(* Logix 5000 project; controller BTS01 vendor 1 type 14 code 217 rev 32.14; software revision 32.04; part 12 of 15 *)
(* tags used below, declared in another part *)
   ApplyDST : SINT;
   C02S03 : INT;   // 5069-IB16
   CAUSTIC_DRAIN_LATCH : BOOL;
   CAUSTIC_DRAIN_RUN : BOOL;
   CAUSTIC_DRAIN_RUN_CLR : BOOL;
   CAUSTIC_DRAIN_RUN_PB : BOOL;
   CAUSTIC_FILL_PB_HMI : BOOL;
   CAUSTIC_FILL_RUN : BOOL;
   CAUSTIC_FILL_RUN_CLR : BOOL;
   CAUSTIC_PREP_LATCH : BOOL;
   CAUSTIC_PREP_RUN : BOOL;
   CAUSTIC_PREP_RUN_CLR : BOOL;   // CAUSTIC PREP JKFF CLEAR BIT
   CAUSTIC_PREP_RUN_PB : BOOL;
   CAUSTIC_PREP_TEMP_SPT : REAL;
   CAUSTIC_PREP_TIME_SPT : REAL;
   CAUSTIC_TANK_LEVEL_OFF_PERC : DINT;   // HMI INPUT OF WATER LEVEL OFF IN %
   CIP1_CAUSTIC_DRAIN_FILE : DINT;   // CIP 1 RAW RECIEVING CIP CAUSTIC DRAIN ENABLE REFERENCE FILE
   CIP1_CAUSTIC_PREP_FILE : DINT;   // CIP 1 RAW RECIEVING CIP CAUSTIC PREP ENABLE REFERENCE FILE
   CIP1_FINALRINSE_DRAIN_FILE : DINT;   // CIP 1 RAW RECIEVING CIP FINAL RINSE DRAIN ENABLE REFERENCE FILE
   CIP1_PRERINSE_DRAIN_FILE : DINT;   // CIP 1 RAW RECIEVING CIP PRERINSE DRAIN ENABLE REFERENCE FILE
   CIP1_PRERINSE_PREP_FILE : DINT;   // CIP 1 RAW RECIEVING CIP PRERINSE PREP ENABLE REFERENCE FILE
   CIP_1_ACTIVE_STEP : CIP_STEP_DEF;   // CIP 1 ACTIVE STEP DATA
   CIP_1_ALARMS : DINT[30];
   CIP_1_AVAIL_STEP_ID : DINT;
   CIP_1_CAUSTIC_TRANS_ACT : BOOL;   // CIP 1 RETURN TO CAUSTIC TANK LEVEL TRANSITION ACTIVE
   CIP_1_CIRCUIT_SELECT_EDIT_HMI : INT;
   CIP_1_EDIT_PROGRAM : CIP_PROGRAM;
   CIP_1_INSERT_STEP : DINT;   // CIP1 INSERT STEP POINTER
   CIP_1_LOAD_RECIPE_EDIT_PB : BOOL;
   CIP_1_MASTER_REF_FILE : DINT[15,30];   // SEQUENCER PINS CIP 1
   CIP_1_PRERINSE_TRANS_ACT : BOOL;   // CIP 1 RETURN TO PRERINSE TANK LEVEL TRANSITION ACTIVE
   CIP_1_PRERINSE_TRANS_DRAIN : BOOL;   // CIP 1 RETURN TO PRERINSE TANK LEVEL TRANSITION ACTIVE
   CIP_1_PROGRAM_ID : INT;
   CIP_1_PROGRAMS : CIP_PROGRAM[30];
   CIP_1_RESET_PB_HMI : BOOL;
   CIP_1_RETURN_HMI : DINT;   // CIP 1 RETURN LOCATION HMI INDICATOR
   CIP_1_RETURN_TO_CAUSTIC : BOOL;   // CIP 1 RETURN TO CAUSTIC TANK DURING CAUSTIC RETURN STEPS
   CIP_1_RETURN_TO_PRERINSE : BOOL;   // CIP 1 RETURN TO PRE-RINSE TANK DURING CAUSTIC RETURN STEPS
   CIP_1_REVERT_RECIPE_EDITS_PB : BOOL;
   CIP_1_RUN_LATCH : BOOL;
   CIP_1_SAVE_RECIPE_EDITS_PB : BOOL;
   CIP_1_SEQ_CTU : COUNTER;   // CIP 1 SEQUENCE STEP COUNTER THIS IS THE SEQUENCE STEP CONTROL
   CIP_1_SEQ_ENABLE : DINT;   // CIP 1 SEQUENCER DATA TO BE ENABLED FOR OPERATION DURING CIP
   CIP_1_STEP_AVAIL_NAMES : CIP_STEP_DEF[30];
   CIP_1_STEP_COPY : BOOL;
   CIP_1_STEP_DELETE : BOOL;
   CIP_1_STEP_DELETING : BOOL;
   CIP_1_STEP_ID : INT;
   CIP_1_STEP_INSERT_PB : BOOL;   // CIP1 STEP INSERT PB FROM HMI
   CIP_1_STEP_INSERTING : BOOL;   // CIP1 STEP INSERTING IN PROGRESS
   CIP_1_TANK_TRANS_VIS_TMR : TIMER;   // CIP 1 TANK TRANSFER VISIBILITY TIMER
   CIP_1_TANK_TRANSITION_HMI : BOOL;   // CIP 1 TANK TRANSITION BANNER VISIBLE ON HMI
   DaylightSavings : Toggle_Bit;
   DTE_TEST : DINT;   // TEST CIP BIT REMOVE WHEN FULL CIP CODE HAS BEEN COMPLETED ==================== Always True Bit
   FINAL_RINSE_DRAIN_LATCH : BOOL;
   FINAL_RINSE_DRAIN_RUN : BOOL;
   FINAL_RINSE_DRAIN_RUN_CLR : BOOL;   // FINAL RINSE JKFF CLEAR BIT
   FINAL_RINSE_DRAIN_RUN_PB : BOOL;
   FINAL_RINSE_FILL_PB_HMI : BOOL;
   FINAL_RINSE_FILL_RUN : BOOL;
   FINAL_RINSE_FILL_RUN_CLR : BOOL;   // FINAL RINSE JKFF CLEAR BIT
   Force_Time_Sync : BOOL;
   LocalTime : DateTime;
   LT351C : Level_Sensor;   // Raw Receiving CIP Pre-Rinse Tank Level Transmitter
   LT352C : Level_Sensor;   // Raw Receiving CIP Caustic Tank Level Transmitter
   LT353C : Level_Sensor;   // Raw Receiving CIP Final Rinse Tank Level Transmitter
   ONS : DINT[20];   // ONE_SHOT_BIT
   PRE_RINSE_TANK_LEVEL_OFF_PERC : DINT;   // HMI INPUT OF WATER LEVEL OFF IN %
   PRERINSE_DRAIN_LATCH : BOOL;
   PRERINSE_DRAIN_RUN : BOOL;
   PRERINSE_DRAIN_RUN_CLR : BOOL;
   PRERINSE_DRAIN_RUN_PB : BOOL;
   PRERINSE_FILL_PB_HMI : BOOL;
   PRERINSE_FILL_RUN : BOOL;
   PRERINSE_FILL_RUN_CLR : BOOL;   // PRE-RINSE FILL JKFF CLEAR BIT
   PRERINSE_PREP_LATCH : BOOL;
   PRERINSE_PREP_RUN : BOOL;
   PRERINSE_PREP_RUN_CLR : BOOL;   // Pre-Rinse Prep JKFF Clear Bit
   PRERINSE_PREP_RUN_PB : BOOL;
   PRERINSE_PREP_TEMP_SPT : REAL;
   PRERINSE_PREP_TIME_SPT : REAL;
   Pulse_DINT : DINT;
   Pulse_LINT : LINT;
   Pulse_Sync_Bit : TIMER;
   Sync_Time_Daily : BOOL;
   TIMERS : TIMER[30];
   Toggle_DST : BOOL;
   TT371C : Temperature_Transmitter;   // Raw Receiving Truck Wash Water Return Temperature Transmitter
(* CIP, continued *)

ROUTINE CIP_Step_Edit   (* ladder *)
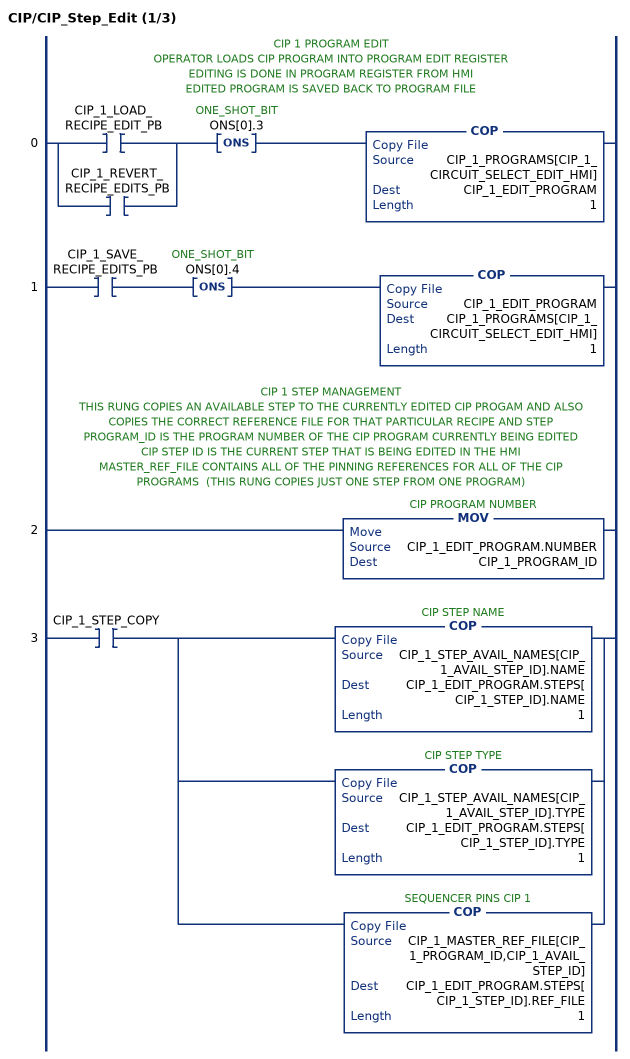
   // CIP 1 PROGRAM EDIT
   // OPERATOR LOADS CIP PROGRAM INTO PROGRAM EDIT REGISTER
   // EDITING IS DONE IN PROGRAM REGISTER FROM HMI
   // EDITED PROGRAM IS SAVED BACK TO PROGRAM FILE
   0: [XIC(CIP_1_LOAD_RECIPE_EDIT_PB) ,XIC(CIP_1_REVERT_RECIPE_EDITS_PB) ]ONS(ONS[0].3)COP(CIP_1_PROGRAMS[CIP_1_CIRCUIT_SELECT_EDIT_HMI],CIP_1_EDIT_PROGRAM,1);
   1: XIC(CIP_1_SAVE_RECIPE_EDITS_PB)ONS(ONS[0].4)COP(CIP_1_EDIT_PROGRAM,CIP_1_PROGRAMS[CIP_1_CIRCUIT_SELECT_EDIT_HMI],1);
   // CIP 1 STEP MANAGEMENT
   // THIS RUNG COPIES AN AVAILABLE STEP TO THE CURRENTLY EDITED CIP PROGAM AND ALSO COPIES THE CORRECT REFERENCE FILE FOR THAT PARTICULAR RECIPE AND STEP
   // PROGRAM_ID IS THE PROGRAM NUMBER OF THE CIP PROGRAM CURRENTLY BEING EDITED
   // CIP STEP ID IS THE CURRENT STEP THAT IS BEING EDITED IN THE HMI
   // MASTER_REF_FILE CONTAINS ALL OF THE PINNING REFERENCES FOR ALL OF THE CIP PROGRAMS  (THIS RUNG COPIES JUST ONE STEP FROM ONE PROGRAM)
   2: MOV(CIP_1_EDIT_PROGRAM.NUMBER,CIP_1_PROGRAM_ID);
   3: XIC(CIP_1_STEP_COPY)[COP(CIP_1_STEP_AVAIL_NAMES[CIP_1_AVAIL_STEP_ID].NAME,CIP_1_EDIT_PROGRAM.STEPS[CIP_1_STEP_ID].NAME,1) ,COP(CIP_1_STEP_AVAIL_NAMES[CIP_1_AVAIL_STEP_ID].TYPE,CIP_1_EDIT_PROGRAM.STEPS[CIP_1_STEP_ID].TYPE,1) ,COP(CIP_1_MASTER_REF_FILE[CIP_1_PROGRAM_ID,CIP_1_AVAIL_STEP_ID],CIP_1_EDIT_PROGRAM.STEPS[CIP_1_STEP_ID].REF_FILE,1) ];
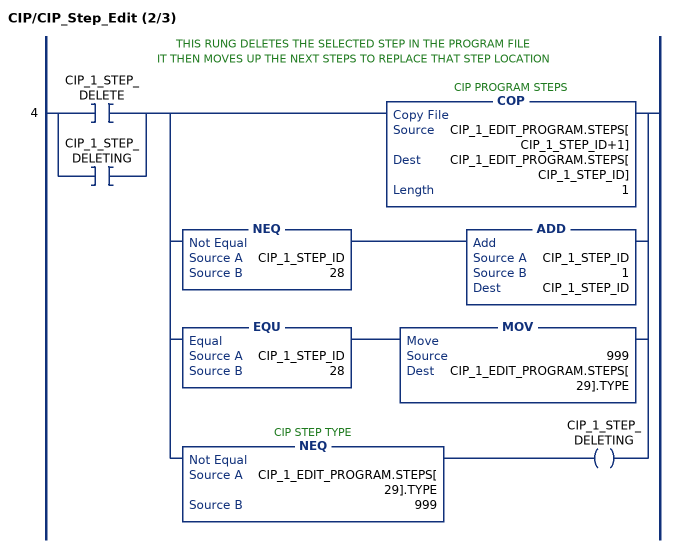
   // THIS RUNG DELETES THE SELECTED STEP IN THE PROGRAM FILE
   // IT THEN MOVES UP THE NEXT STEPS TO REPLACE THAT STEP LOCATION
   4: [XIC(CIP_1_STEP_DELETE) ,XIC(CIP_1_STEP_DELETING) ][COP(CIP_1_EDIT_PROGRAM.STEPS[CIP_1_STEP_ID+1],CIP_1_EDIT_PROGRAM.STEPS[CIP_1_STEP_ID],1) ,NEQ(CIP_1_STEP_ID,28) ADD(CIP_1_STEP_ID,1,CIP_1_STEP_ID) ,EQU(CIP_1_STEP_ID,28) MOV(999,CIP_1_EDIT_PROGRAM.STEPS[29].TYPE) ,NEQ(CIP_1_EDIT_PROGRAM.STEPS[29].TYPE,999) OTE(CIP_1_STEP_DELETING) ];
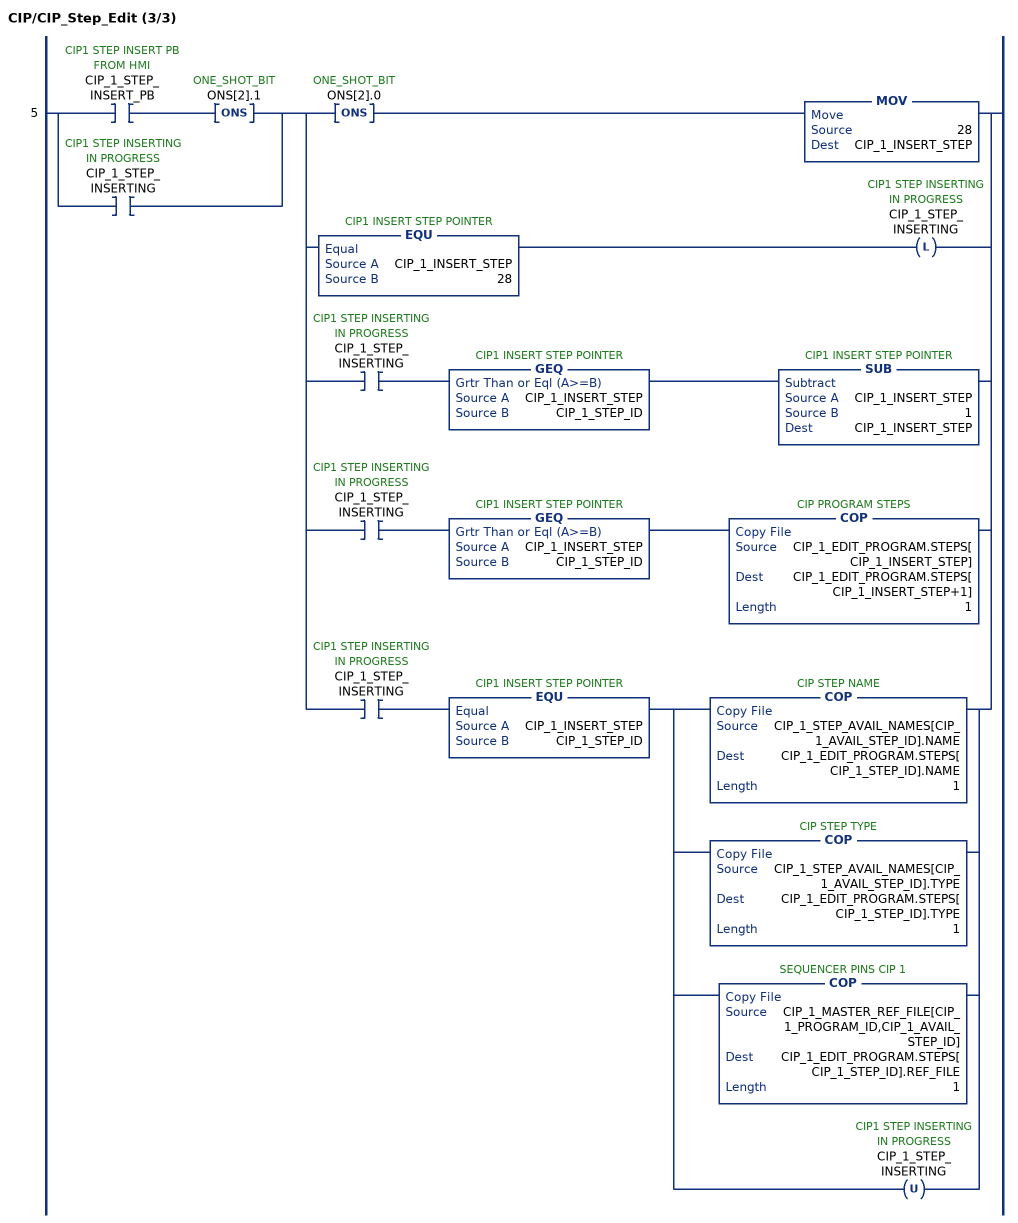
   5: [XIC(CIP_1_STEP_INSERT_PB) ONS(ONS[2].1) ,XIC(CIP_1_STEP_INSERTING) ][ONS(ONS[2].0) MOV(28,CIP_1_INSERT_STEP) ,EQU(CIP_1_INSERT_STEP,28) OTL(CIP_1_STEP_INSERTING) ,XIC(CIP_1_STEP_INSERTING) GEQ(CIP_1_INSERT_STEP,CIP_1_STEP_ID) SUB(CIP_1_INSERT_STEP,1,CIP_1_INSERT_STEP) ,XIC(CIP_1_STEP_INSERTING) GEQ(CIP_1_INSERT_STEP,CIP_1_STEP_ID) COP(CIP_1_EDIT_PROGRAM.STEPS[CIP_1_INSERT_STEP],CIP_1_EDIT_PROGRAM.STEPS[CIP_1_INSERT_STEP+1],1) ,XIC(CIP_1_STEP_INSERTING) EQU(CIP_1_INSERT_STEP,CIP_1_STEP_ID) [COP(CIP_1_STEP_AVAIL_NAMES[CIP_1_AVAIL_STEP_ID].NAME,CIP_1_EDIT_PROGRAM.STEPS[CIP_1_STEP_ID].NAME,1) ,COP(CIP_1_STEP_AVAIL_NAMES[CIP_1_AVAIL_STEP_ID].TYPE,CIP_1_EDIT_PROGRAM.STEPS[CIP_1_STEP_ID].TYPE,1) ,COP(CIP_1_MASTER_REF_FILE[CIP_1_PROGRAM_ID,CIP_1_AVAIL_STEP_ID],CIP_1_EDIT_PROGRAM.STEPS[CIP_1_STEP_ID].REF_FILE,1) ,OTU(CIP_1_STEP_INSERTING) ] ];
END_ROUTINE

ROUTINE CIP_Tank_Transition   (* ladder *)
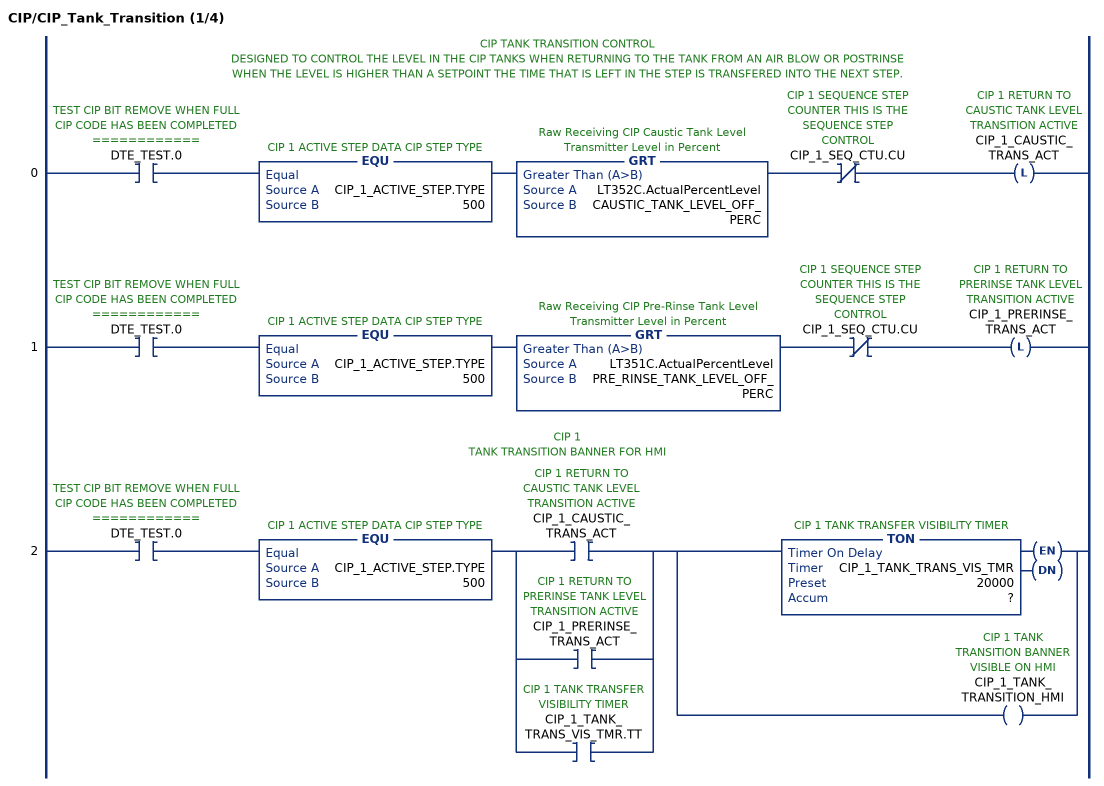
   // CIP TANK TRANSITION CONTROL
   // DESIGNED TO CONTROL THE LEVEL IN THE CIP TANKS WHEN RETURNING TO THE TANK FROM AN AIR BLOW OR POSTRINSE
   // WHEN THE LEVEL IS HIGHER THAN A SETPOINT THE TIME THAT IS LEFT IN THE STEP IS TRANSFERED INTO THE NEXT STEP.
   0: XIC(DTE_TEST.0)EQU(CIP_1_ACTIVE_STEP.TYPE,500)GRT(LT352C.ActualPercentLevel,CAUSTIC_TANK_LEVEL_OFF_PERC)XIO(CIP_1_SEQ_CTU.CU)OTL(CIP_1_CAUSTIC_TRANS_ACT);
   1: XIC(DTE_TEST.0)EQU(CIP_1_ACTIVE_STEP.TYPE,500)GRT(LT351C.ActualPercentLevel,PRE_RINSE_TANK_LEVEL_OFF_PERC)XIO(CIP_1_SEQ_CTU.CU)OTL(CIP_1_PRERINSE_TRANS_ACT);
   // CIP 1
   // TANK TRANSITION BANNER FOR HMI
   2: XIC(DTE_TEST.0)EQU(CIP_1_ACTIVE_STEP.TYPE,500)[XIC(CIP_1_CAUSTIC_TRANS_ACT) ,XIC(CIP_1_PRERINSE_TRANS_ACT) ,XIC(CIP_1_TANK_TRANS_VIS_TMR.TT) ][TON(CIP_1_TANK_TRANS_VIS_TMR,?,?) ,OTE(CIP_1_TANK_TRANSITION_HMI) ];
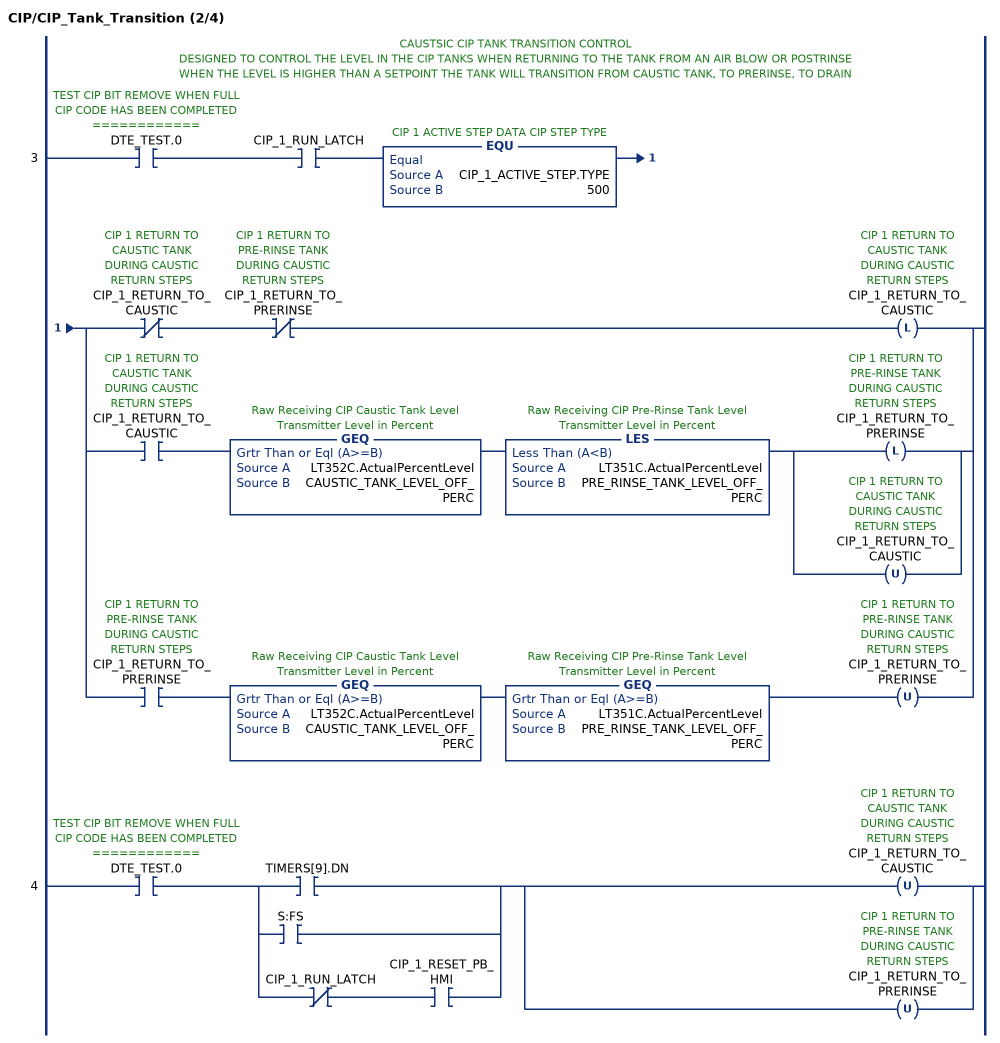
   // CAUSTSIC CIP TANK TRANSITION CONTROL
   // DESIGNED TO CONTROL THE LEVEL IN THE CIP TANKS WHEN RETURNING TO THE TANK FROM AN AIR BLOW OR POSTRINSE
   // WHEN THE LEVEL IS HIGHER THAN A SETPOINT THE TANK WILL TRANSITION FROM CAUSTIC TANK, TO PRERINSE, TO DRAIN
   3: XIC(DTE_TEST.0)XIC(CIP_1_RUN_LATCH)EQU(CIP_1_ACTIVE_STEP.TYPE,500)[XIO(CIP_1_RETURN_TO_CAUSTIC) XIO(CIP_1_RETURN_TO_PRERINSE) OTL(CIP_1_RETURN_TO_CAUSTIC) ,XIC(CIP_1_RETURN_TO_CAUSTIC) GEQ(LT352C.ActualPercentLevel,CAUSTIC_TANK_LEVEL_OFF_PERC) LES(LT351C.ActualPercentLevel,PRE_RINSE_TANK_LEVEL_OFF_PERC) [OTL(CIP_1_RETURN_TO_PRERINSE) ,OTU(CIP_1_RETURN_TO_CAUSTIC) ] ,XIC(CIP_1_RETURN_TO_PRERINSE) GEQ(LT352C.ActualPercentLevel,CAUSTIC_TANK_LEVEL_OFF_PERC) GEQ(LT351C.ActualPercentLevel,PRE_RINSE_TANK_LEVEL_OFF_PERC) OTU(CIP_1_RETURN_TO_PRERINSE) ];
   4: XIC(DTE_TEST.0)[XIC(TIMERS[9].DN) ,XIC(S:FS) ,XIO(CIP_1_RUN_LATCH) XIC(CIP_1_RESET_PB_HMI) ][OTU(CIP_1_RETURN_TO_CAUSTIC) ,OTU(CIP_1_RETURN_TO_PRERINSE) ];
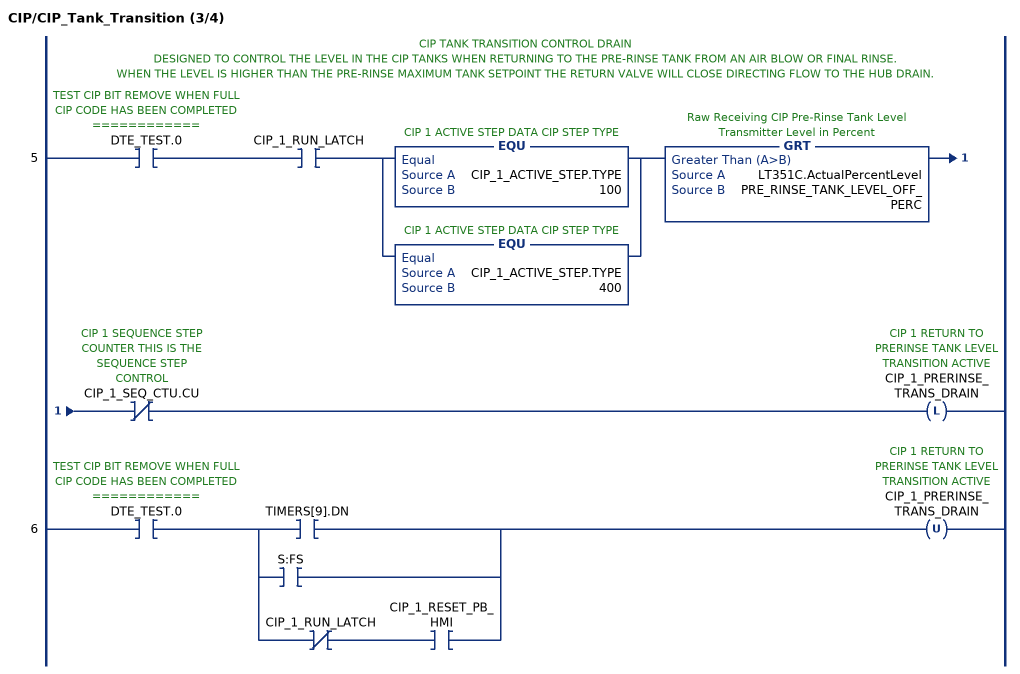
   // CIP TANK TRANSITION CONTROL DRAIN
   // DESIGNED TO CONTROL THE LEVEL IN THE CIP TANKS WHEN RETURNING TO THE PRE-RINSE TANK FROM AN AIR BLOW OR FINAL RINSE.
   // WHEN THE LEVEL IS HIGHER THAN THE PRE-RINSE MAXIMUM TANK SETPOINT THE RETURN VALVE WILL CLOSE DIRECTING FLOW TO THE HUB DRAIN.
   5: XIC(DTE_TEST.0)XIC(CIP_1_RUN_LATCH)[EQU(CIP_1_ACTIVE_STEP.TYPE,100) ,EQU(CIP_1_ACTIVE_STEP.TYPE,400) ]GRT(LT351C.ActualPercentLevel,PRE_RINSE_TANK_LEVEL_OFF_PERC)XIO(CIP_1_SEQ_CTU.CU)OTL(CIP_1_PRERINSE_TRANS_DRAIN);
   6: XIC(DTE_TEST.0)[XIC(TIMERS[9].DN) ,XIC(S:FS) ,XIO(CIP_1_RUN_LATCH) XIC(CIP_1_RESET_PB_HMI) ]OTU(CIP_1_PRERINSE_TRANS_DRAIN);
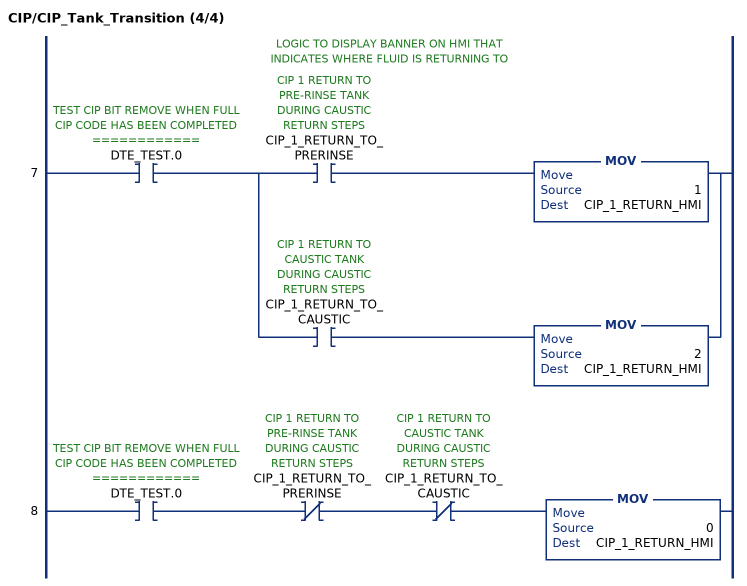
   // LOGIC TO DISPLAY BANNER ON HMI THAT
   // INDICATES WHERE FLUID IS RETURNING TO
   7: XIC(DTE_TEST.0)[XIC(CIP_1_RETURN_TO_PRERINSE) MOV(1,CIP_1_RETURN_HMI) ,XIC(CIP_1_RETURN_TO_CAUSTIC) MOV(2,CIP_1_RETURN_HMI) ];
   8: XIC(DTE_TEST.0)XIO(CIP_1_RETURN_TO_PRERINSE)XIO(CIP_1_RETURN_TO_CAUSTIC)MOV(0,CIP_1_RETURN_HMI);
END_ROUTINE

ROUTINE Drain_Prep_Functions   (* ladder *)
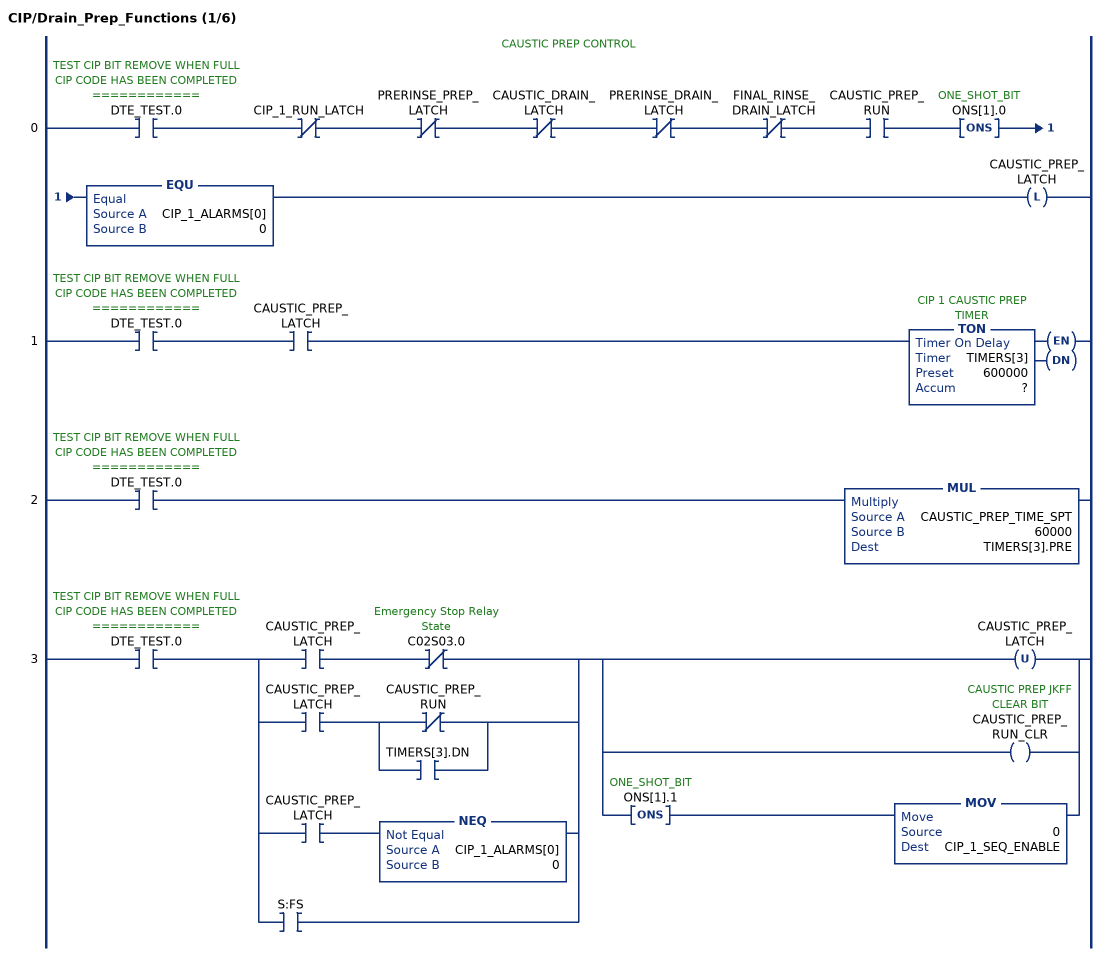
   // CAUSTIC PREP CONTROL
   0: XIC(DTE_TEST.0)XIO(CIP_1_RUN_LATCH)XIO(PRERINSE_PREP_LATCH)XIO(CAUSTIC_DRAIN_LATCH)XIO(PRERINSE_DRAIN_LATCH)XIO(FINAL_RINSE_DRAIN_LATCH)XIC(CAUSTIC_PREP_RUN)ONS(ONS[1].0)EQU(CIP_1_ALARMS[0],0)OTL(CAUSTIC_PREP_LATCH);
   1: XIC(DTE_TEST.0)XIC(CAUSTIC_PREP_LATCH)TON(TIMERS[3],?,?);
   2: XIC(DTE_TEST.0)MUL(CAUSTIC_PREP_TIME_SPT,60000,TIMERS[3].PRE);
   3: XIC(DTE_TEST.0)[XIC(CAUSTIC_PREP_LATCH) XIO(C02S03.0) ,XIC(CAUSTIC_PREP_LATCH) [XIO(CAUSTIC_PREP_RUN) ,XIC(TIMERS[3].DN) ] ,XIC(CAUSTIC_PREP_LATCH) NEQ(CIP_1_ALARMS[0],0) ,XIC(S:FS) ][OTU(CAUSTIC_PREP_LATCH) ,OTE(CAUSTIC_PREP_RUN_CLR) ,ONS(ONS[1].1) MOV(0,CIP_1_SEQ_ENABLE) ];
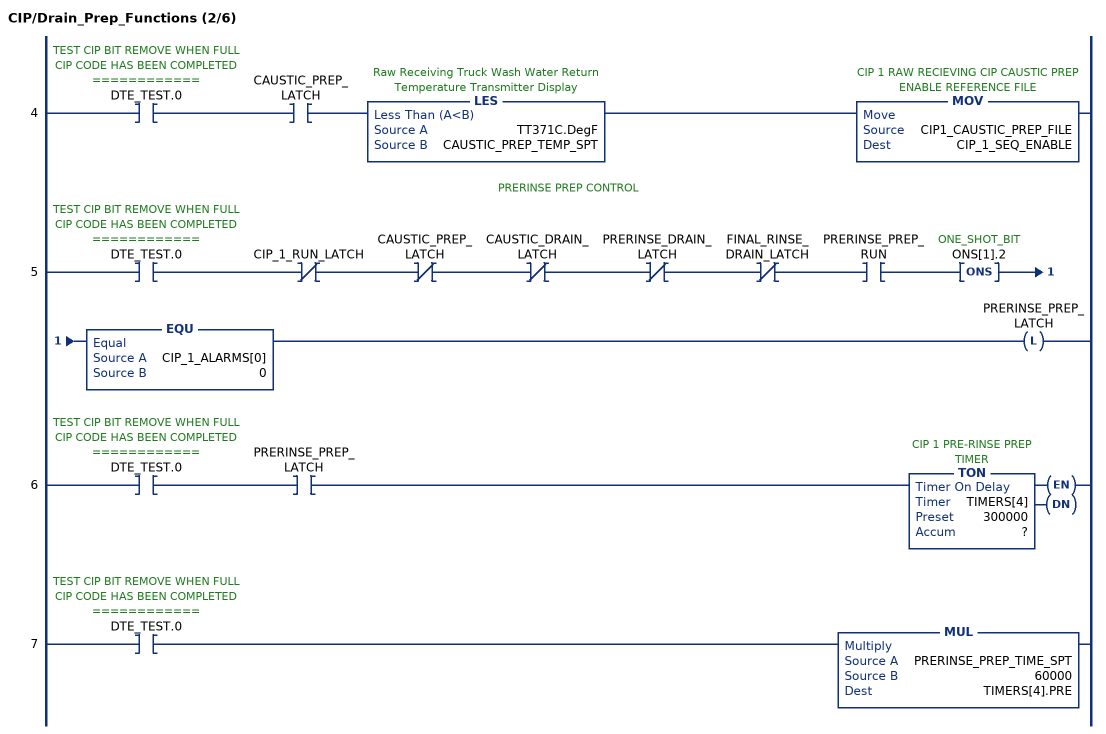
   4: XIC(DTE_TEST.0)XIC(CAUSTIC_PREP_LATCH)LES(TT371C.DegF,CAUSTIC_PREP_TEMP_SPT)MOV(CIP1_CAUSTIC_PREP_FILE,CIP_1_SEQ_ENABLE);
   // PRERINSE PREP CONTROL
   5: XIC(DTE_TEST.0)XIO(CIP_1_RUN_LATCH)XIO(CAUSTIC_PREP_LATCH)XIO(CAUSTIC_DRAIN_LATCH)XIO(PRERINSE_DRAIN_LATCH)XIO(FINAL_RINSE_DRAIN_LATCH)XIC(PRERINSE_PREP_RUN)ONS(ONS[1].2)EQU(CIP_1_ALARMS[0],0)OTL(PRERINSE_PREP_LATCH);
   6: XIC(DTE_TEST.0)XIC(PRERINSE_PREP_LATCH)TON(TIMERS[4],?,?);
   7: XIC(DTE_TEST.0)MUL(PRERINSE_PREP_TIME_SPT,60000,TIMERS[4].PRE);
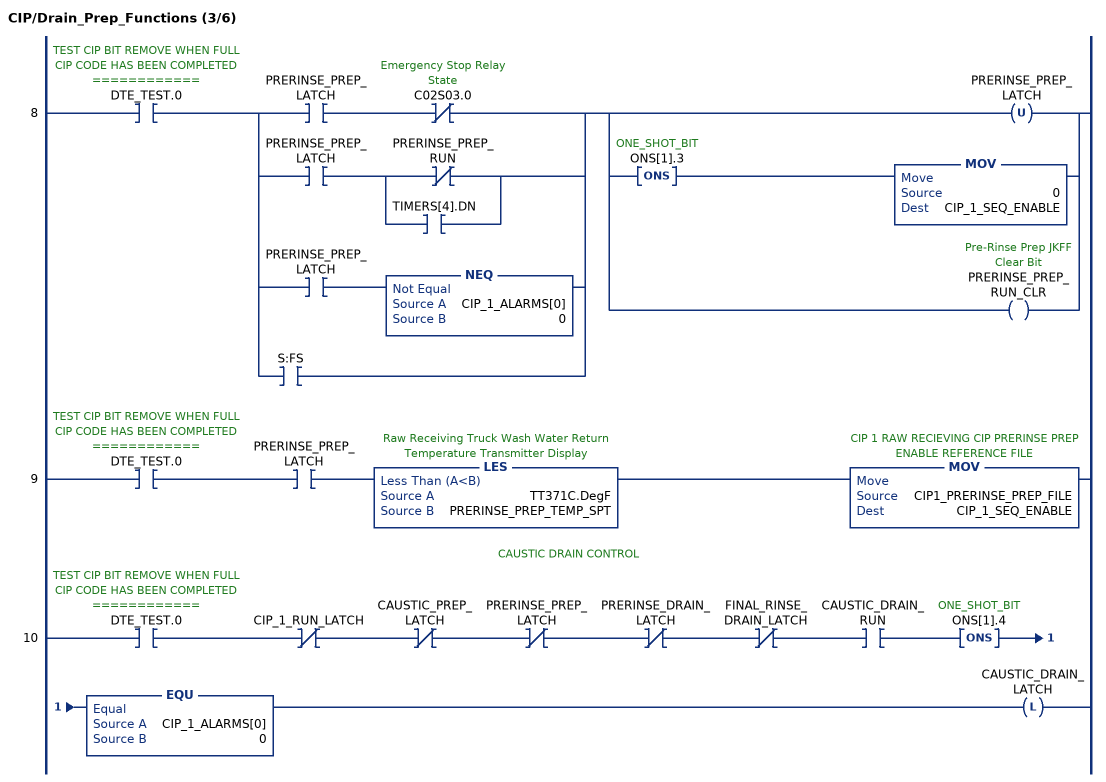
   8: XIC(DTE_TEST.0)[XIC(PRERINSE_PREP_LATCH) XIO(C02S03.0) ,XIC(PRERINSE_PREP_LATCH) [XIO(PRERINSE_PREP_RUN) ,XIC(TIMERS[4].DN) ] ,XIC(PRERINSE_PREP_LATCH) NEQ(CIP_1_ALARMS[0],0) ,XIC(S:FS) ][OTU(PRERINSE_PREP_LATCH) ,ONS(ONS[1].3) MOV(0,CIP_1_SEQ_ENABLE) ,OTE(PRERINSE_PREP_RUN_CLR) ];
   9: XIC(DTE_TEST.0)XIC(PRERINSE_PREP_LATCH)LES(TT371C.DegF,PRERINSE_PREP_TEMP_SPT)MOV(CIP1_PRERINSE_PREP_FILE,CIP_1_SEQ_ENABLE);
   // CAUSTIC DRAIN CONTROL
   10: XIC(DTE_TEST.0)XIO(CIP_1_RUN_LATCH)XIO(CAUSTIC_PREP_LATCH)XIO(PRERINSE_PREP_LATCH)XIO(PRERINSE_DRAIN_LATCH)XIO(FINAL_RINSE_DRAIN_LATCH)XIC(CAUSTIC_DRAIN_RUN)ONS(ONS[1].4)EQU(CIP_1_ALARMS[0],0)OTL(CAUSTIC_DRAIN_LATCH);
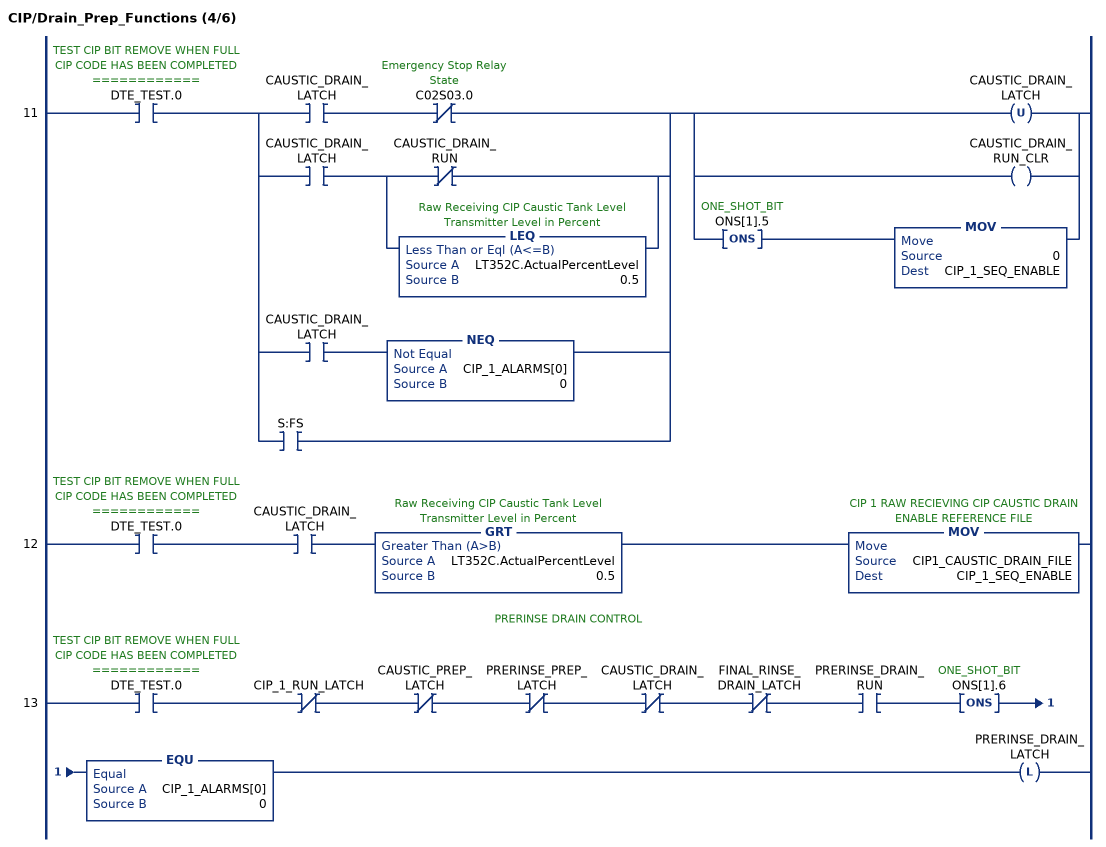
   11: XIC(DTE_TEST.0)[XIC(CAUSTIC_DRAIN_LATCH) XIO(C02S03.0) ,XIC(CAUSTIC_DRAIN_LATCH) [XIO(CAUSTIC_DRAIN_RUN) ,LEQ(LT352C.ActualPercentLevel,0.5) ] ,XIC(CAUSTIC_DRAIN_LATCH) NEQ(CIP_1_ALARMS[0],0) ,XIC(S:FS) ][OTU(CAUSTIC_DRAIN_LATCH) ,OTE(CAUSTIC_DRAIN_RUN_CLR) ,ONS(ONS[1].5) MOV(0,CIP_1_SEQ_ENABLE) ];
   12: XIC(DTE_TEST.0)XIC(CAUSTIC_DRAIN_LATCH)GRT(LT352C.ActualPercentLevel,0.5)MOV(CIP1_CAUSTIC_DRAIN_FILE,CIP_1_SEQ_ENABLE);
   // PRERINSE DRAIN CONTROL
   13: XIC(DTE_TEST.0)XIO(CIP_1_RUN_LATCH)XIO(CAUSTIC_PREP_LATCH)XIO(PRERINSE_PREP_LATCH)XIO(CAUSTIC_DRAIN_LATCH)XIO(FINAL_RINSE_DRAIN_LATCH)XIC(PRERINSE_DRAIN_RUN)ONS(ONS[1].6)EQU(CIP_1_ALARMS[0],0)OTL(PRERINSE_DRAIN_LATCH);
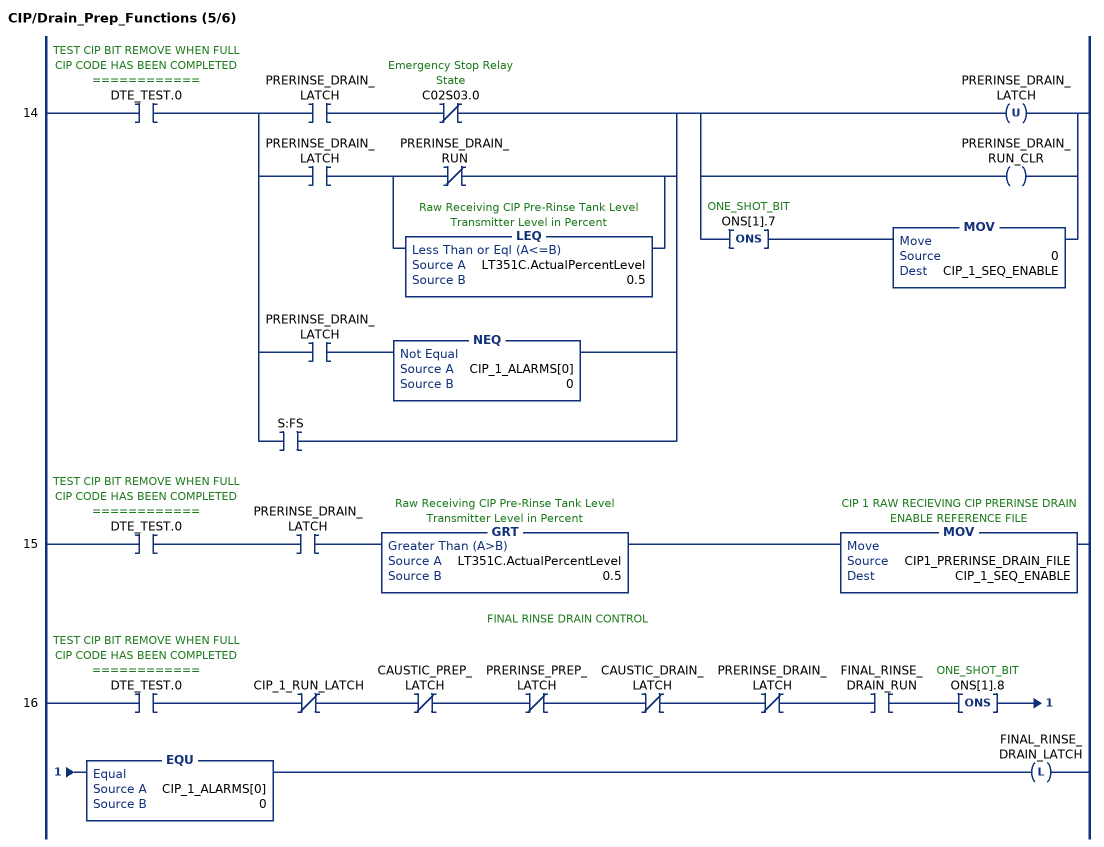
   14: XIC(DTE_TEST.0)[XIC(PRERINSE_DRAIN_LATCH) XIO(C02S03.0) ,XIC(PRERINSE_DRAIN_LATCH) [XIO(PRERINSE_DRAIN_RUN) ,LEQ(LT351C.ActualPercentLevel,0.5) ] ,XIC(PRERINSE_DRAIN_LATCH) NEQ(CIP_1_ALARMS[0],0) ,XIC(S:FS) ][OTU(PRERINSE_DRAIN_LATCH) ,OTE(PRERINSE_DRAIN_RUN_CLR) ,ONS(ONS[1].7) MOV(0,CIP_1_SEQ_ENABLE) ];
   15: XIC(DTE_TEST.0)XIC(PRERINSE_DRAIN_LATCH)GRT(LT351C.ActualPercentLevel,0.5)MOV(CIP1_PRERINSE_DRAIN_FILE,CIP_1_SEQ_ENABLE);
   // FINAL RINSE DRAIN CONTROL
   16: XIC(DTE_TEST.0)XIO(CIP_1_RUN_LATCH)XIO(CAUSTIC_PREP_LATCH)XIO(PRERINSE_PREP_LATCH)XIO(CAUSTIC_DRAIN_LATCH)XIO(PRERINSE_DRAIN_LATCH)XIC(FINAL_RINSE_DRAIN_RUN)ONS(ONS[1].8)EQU(CIP_1_ALARMS[0],0)OTL(FINAL_RINSE_DRAIN_LATCH);
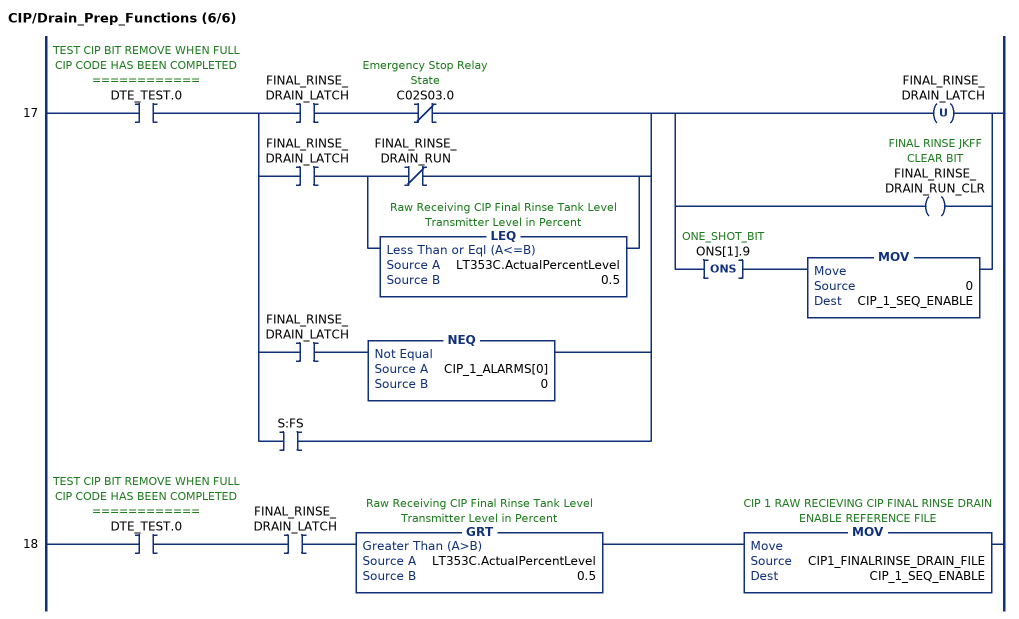
   17: XIC(DTE_TEST.0)[XIC(FINAL_RINSE_DRAIN_LATCH) XIO(C02S03.0) ,XIC(FINAL_RINSE_DRAIN_LATCH) [XIO(FINAL_RINSE_DRAIN_RUN) ,LEQ(LT353C.ActualPercentLevel,0.5) ] ,XIC(FINAL_RINSE_DRAIN_LATCH) NEQ(CIP_1_ALARMS[0],0) ,XIC(S:FS) ][OTU(FINAL_RINSE_DRAIN_LATCH) ,OTE(FINAL_RINSE_DRAIN_RUN_CLR) ,ONS(ONS[1].9) MOV(0,CIP_1_SEQ_ENABLE) ];
   18: XIC(DTE_TEST.0)XIC(FINAL_RINSE_DRAIN_LATCH)GRT(LT353C.ActualPercentLevel,0.5)MOV(CIP1_FINALRINSE_DRAIN_FILE,CIP_1_SEQ_ENABLE);
END_ROUTINE

ROUTINE Main_Routine   (* ladder *)
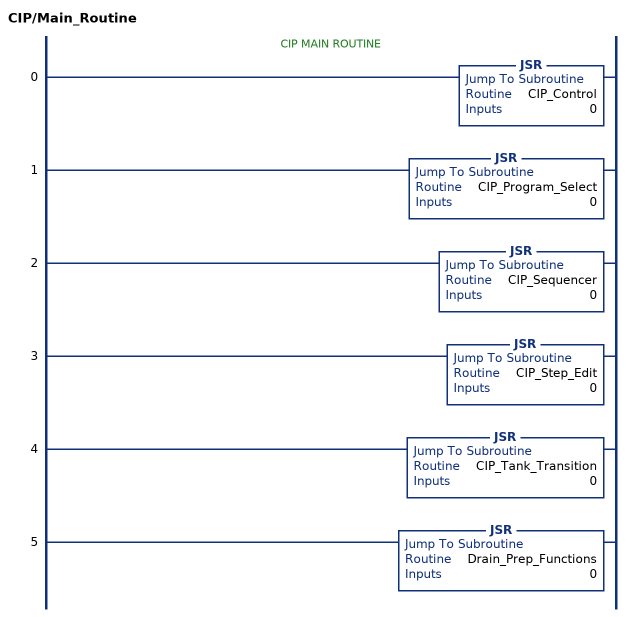
   // CIP MAIN ROUTINE
   0: JSR(CIP_Control,0);
   1: JSR(CIP_Program_Select,0);
   2: JSR(CIP_Sequencer,0);
   3: JSR(CIP_Step_Edit,0);
   4: JSR(CIP_Tank_Transition,0);
   5: JSR(Drain_Prep_Functions,0);
END_ROUTINE
END_PROGRAM

PROGRAM MainProgram   (* main routine MainRoutine *)
VAR
   CAUSTIC_DRAIN : FLIP_FLOP_JK := (QNot := 1);
   CAUSTIC_FILL : FLIP_FLOP_JK := (QNot := 1);
   CAUSTIC_PREP : FLIP_FLOP_JK := (QNot := 1);
   FINAL_RINSE_DRAIN : FLIP_FLOP_JK := (QNot := 1);
   FINAL_RINSE_FILL : FLIP_FLOP_JK := (QNot := 1);
   PRERINSE_DRAIN : FLIP_FLOP_JK := (QNot := 1);
   PRERINSE_FILL : FLIP_FLOP_JK := (QNot := 1);
   PRERINSE_PREP : FLIP_FLOP_JK := (QNot := 1);
END_VAR

ROUTINE HMI_Pushbuttons   (* function block diagram *)
   SHEET 1
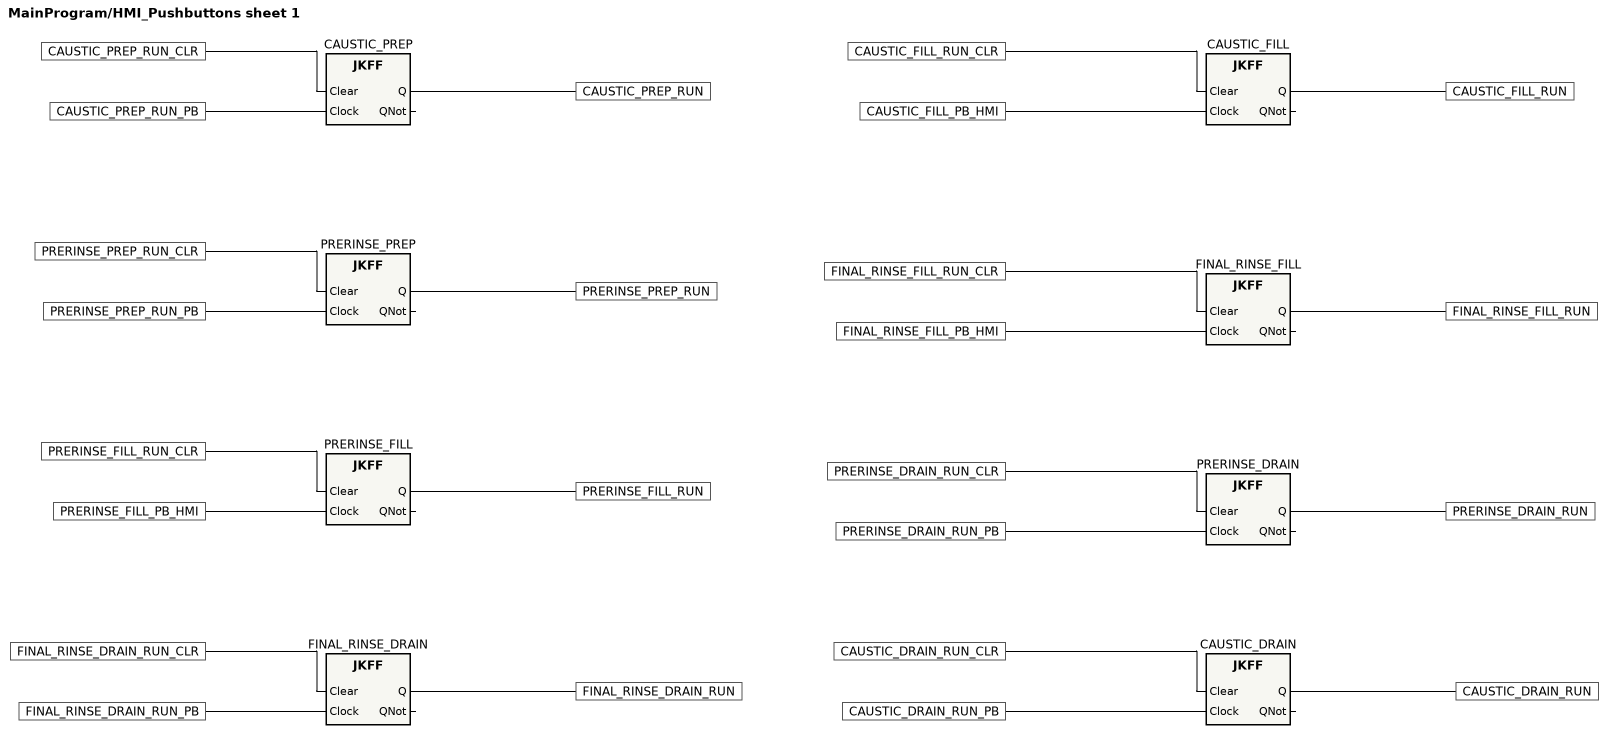
   CAUSTIC_PREP : JKFF(Clear := CAUSTIC_PREP_RUN_CLR, Clock := CAUSTIC_PREP_RUN_PB);   // unwired pins: QNot
   PRERINSE_PREP : JKFF(Clear := PRERINSE_PREP_RUN_CLR, Clock := PRERINSE_PREP_RUN_PB);   // unwired pins: QNot
   PRERINSE_FILL : JKFF(Clear := PRERINSE_FILL_RUN_CLR, Clock := PRERINSE_FILL_PB_HMI);   // unwired pins: QNot
   FINAL_RINSE_DRAIN : JKFF(Clear := FINAL_RINSE_DRAIN_RUN_CLR, Clock := FINAL_RINSE_DRAIN_RUN_PB);   // unwired pins: QNot
   CAUSTIC_PREP_RUN := CAUSTIC_PREP.Q;
   PRERINSE_PREP_RUN := PRERINSE_PREP.Q;
   PRERINSE_FILL_RUN := PRERINSE_FILL.Q;
   FINAL_RINSE_DRAIN_RUN := FINAL_RINSE_DRAIN.Q;
   CAUSTIC_FILL : JKFF(Clear := CAUSTIC_FILL_RUN_CLR, Clock := CAUSTIC_FILL_PB_HMI);   // unwired pins: QNot
   FINAL_RINSE_FILL : JKFF(Clear := FINAL_RINSE_FILL_RUN_CLR, Clock := FINAL_RINSE_FILL_PB_HMI);   // unwired pins: QNot
   PRERINSE_DRAIN : JKFF(Clear := PRERINSE_DRAIN_RUN_CLR, Clock := PRERINSE_DRAIN_RUN_PB);   // unwired pins: QNot
   CAUSTIC_DRAIN : JKFF(Clear := CAUSTIC_DRAIN_RUN_CLR, Clock := CAUSTIC_DRAIN_RUN_PB);   // unwired pins: QNot
   CAUSTIC_FILL_RUN := CAUSTIC_FILL.Q;
   FINAL_RINSE_FILL_RUN := FINAL_RINSE_FILL.Q;
   PRERINSE_DRAIN_RUN := PRERINSE_DRAIN.Q;
   CAUSTIC_DRAIN_RUN := CAUSTIC_DRAIN.Q;
END_ROUTINE

ROUTINE MainRoutine   (* ladder *)
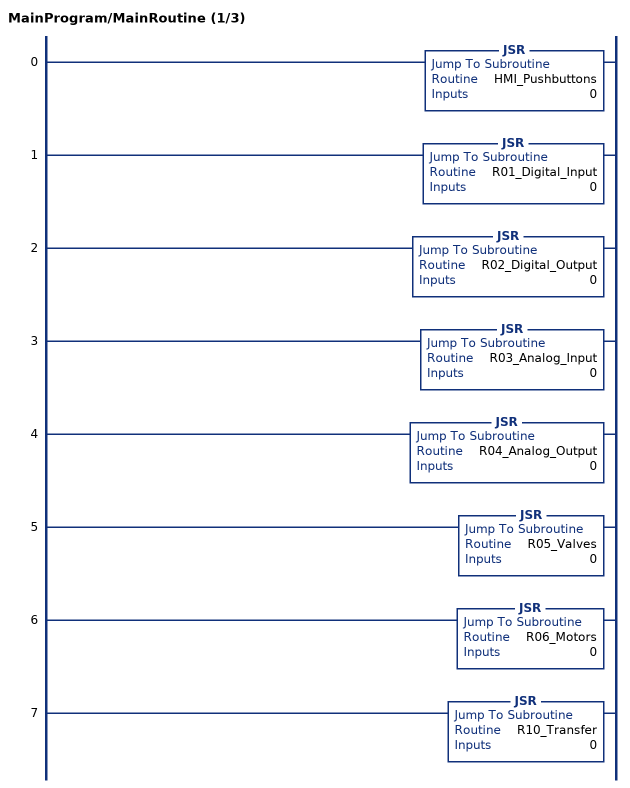
   0: JSR(HMI_Pushbuttons,0);
   1: JSR(R01_Digital_Input,0);
   2: JSR(R02_Digital_Output,0);
   3: JSR(R03_Analog_Input,0);
   4: JSR(R04_Analog_Output,0);
   5: JSR(R05_Valves,0);
   6: JSR(R06_Motors,0);
   7: JSR(R10_Transfer,0);
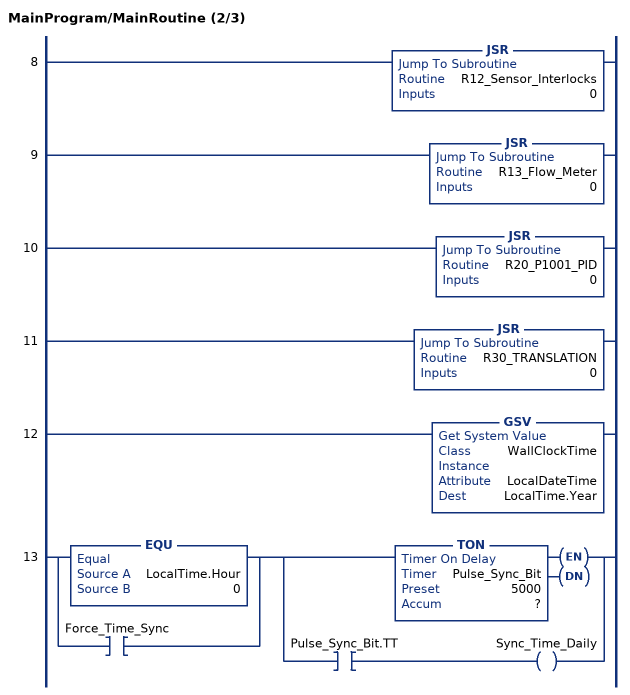
   8: JSR(R12_Sensor_Interlocks,0);
   9: JSR(R13_Flow_Meter,0);
   10: JSR(R20_P1001_PID,0);
   11: JSR(R30_TRANSLATION,0);
   12: GSV(WallClockTime,,LocalDateTime,LocalTime.Year);
   13: [EQU(LocalTime.Hour,0) ,XIC(Force_Time_Sync) ][TON(Pulse_Sync_Bit,?,?) ,XIC(Pulse_Sync_Bit.TT) OTE(Sync_Time_Daily) ];
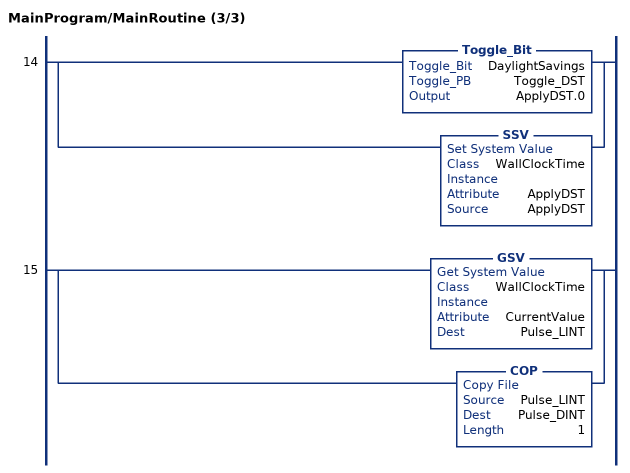
   14: [Toggle_Bit(DaylightSavings,Toggle_DST,ApplyDST.0) ,SSV(WallClockTime,,ApplyDST,ApplyDST) ];
   15: [GSV(WallClockTime,,CurrentValue,Pulse_LINT) ,COP(Pulse_LINT,Pulse_DINT,1) ];
END_ROUTINE
